{attribute 'qualified_only'}
VAR_GLOBAL
		EtherCAT_Master_ERxxxx : EtherCAT_Master_ERxxxx_3A895043;
END_VAR

(* stored: Version 1.2.0.0, ProductVersion 3.1.4024.9
   GVL GVL_iXlinker: Id {cd92dcac-23d5-40c6-b3cc-292957d23fc9} *)
